KUKA KRL program: style1drop1opt2AutoRR.src, style1drop1opt2AutoRR.dat

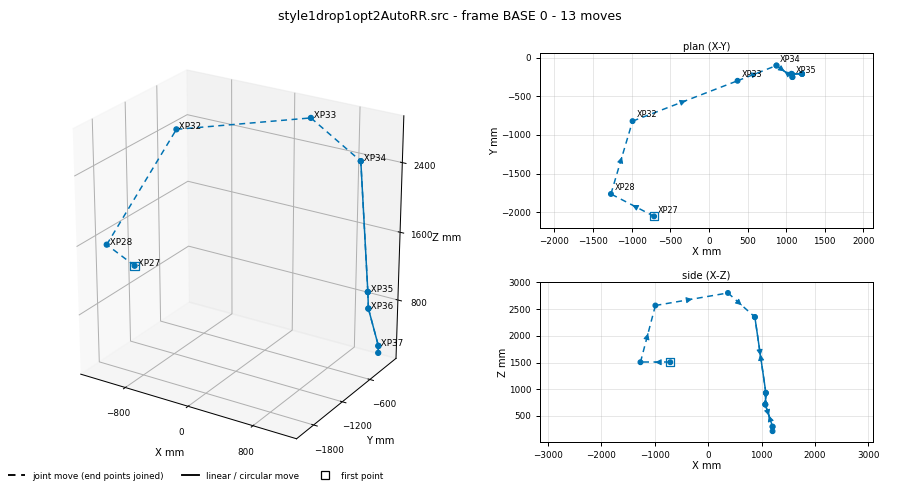
[picture p0: tool path of style1drop1opt2AutoRR.src in frame BASE 0, 13 of 14 moves have a stored position in this frame; points joined in program order, loops and branches not executed]
--- style1drop1opt2AutoRR.src ---
&ACCESS RVO1
&REL 269
&COMMENT 03-10-R1 RED RABBIT DROP
&PARAM EDITMASK = *
&PARAM DISKPATH = KRC:\R1\Program\StyleDrops\Options
DEF style1drop1opt2AutoRR( )
   ;FOLD INI
      ;FOLD BASISTECH INI
         GLOBAL INTERRUPT DECL 3 WHEN $STOPMESS==TRUE DO IR_STOPM ( )
         INTERRUPT ON 3
         BAS (#INITMOV,0 )
      ;ENDFOLD (BASISTECH INI)
      ;FOLD USER INI
         ;Make your modifications here

      ;ENDFOLD (USER INI)
   ;ENDFOLD (INI)
;********************************
; Gestamp Standards
; Line - BMW G65 (cell 03)
; Robot 03-10-R1 (BMW-03-10-R1-MH1)
; Application - RED RABBIT DROP AT DROPOFF 2
;********************************
; CALLED BY Style1Opt10AutoRR (OPTION 12). TAKES THE RED RABBIT PART TO AtPick3 OF THIS MODULE
; AND RELEASES IT, THEN CLEARS THE RED RABBIT OUTPUTS AND THE NUT FLAGS AND RETURNS HOME.
;WARNING: GRIPPER 1 IS DRIVEN TO CLOSE AT THE START ($OUT[250] ON) AND THE RELEASE COMMAND
;  OPENS GRIPPER 3, WHICH IS INACTIVE IN grp_data.dat: GRIPPER 1 DOES NOT OPEN, THE CHECK OF
;  GRIPPER 1 OPEN THAT FOLLOWS FAILS (F19, F31)
;NOTE: THE ROBOT MOVES AWAY (LIN P23) BEFORE THE GRIPPER-EMPTY WAIT (F40)
;DROPOFF 2 REQUEST - AC_DropOffCheck(2): WAIT SIGNAL $IN[76] di076DropOffMachine2 ON
;(WAITING MESSAGE, NO TIMEOUT), THEN SIGNALS $OUT[76] do076DropOffClear2 OFF,
;$OUT[25] do025DropClearTooling OFF
;FOLD DropOff[2] Request
;FOLD ;%{h}
;Params IlfProvider=ac_zoneilf; AC_CmdZones=DropOff; AC_CmdParam=2; AC_ZoneRepo=False; AC_Blending=False
;ENDFOLD
AC_DropOffCheck (2)
;ENDFOLD

;GRIPPER 1 CLOSE (HAND-WRITTEN OUTPUTS, NO CHECK) - SIGNALS $OUT[249] do249Group1Home OFF,
;$OUT[250] do250Group1Work ON (CONTINUE: SET IN THE ADVANCE RUN)
;FOLD OUT 249 'do249Group1Home' State=FALSE CONT;%{PE}%R 8.3.43,%MKUKATPBASIS,%COUT,%VOUTX,%P 2:249, 3:do249Group1Home, 5:FALSE, 6:CONTINUE
CONTINUE
$OUT[249]=FALSE
;ENDFOLD
;FOLD OUT 250 'do250Group1Work' State=TRUE CONT;%{PE}%R 8.3.43,%MKUKATPBASIS,%COUT,%VOUTX,%P 2:250, 3:do250Group1Work, 5:TRUE, 6:CONTINUE
CONTINUE
$OUT[250]=TRUE
;ENDFOLD

;APPROACH THE RED RABBIT DROP - P27, P28, P32, P33, P34, P35, P36, P37, AtPick3
;FOLD PTP P27 Vel=100 % PDAT25 Tool[1]:TOOL 1 Base[0];%{PE}%R 8.3.43,%MKUKATPBASIS,%CMOVE,%VPTP,%P 1:PTP, 2:P27, 3:, 5:100, 7:PDAT25
$BWDSTART=FALSE
PDAT_ACT=PPDAT25
FDAT_ACT=FP27
BAS(#PTP_PARAMS,100)
PTP XP27
;ENDFOLD
;FOLD PTP P28 Vel=100 % PDAT26 Tool[1]:TOOL 1 Base[0];%{PE}%R 8.3.43,%MKUKATPBASIS,%CMOVE,%VPTP,%P 1:PTP, 2:P28, 3:, 5:100, 7:PDAT26
$BWDSTART=FALSE
PDAT_ACT=PPDAT26
FDAT_ACT=FP28
BAS(#PTP_PARAMS,100)
PTP XP28
;ENDFOLD


;FOLD PTP P32 CONT Vel=100 % PDAT30 Tool[1]:TOOL 1 Base[0];%{PE}%R 8.3.43,%MKUKATPBASIS,%CMOVE,%VPTP,%P 1:PTP, 2:P32, 3:C_DIS, 5:100, 7:PDAT30
$BWDSTART=FALSE
PDAT_ACT=PPDAT30
FDAT_ACT=FP32
BAS(#PTP_PARAMS,100)
PTP XP32 C_DIS
;ENDFOLD
;FOLD PTP P33 Vel=100 % PDAT31 Tool[1]:TOOL 1 Base[0];%{PE}%R 8.3.43,%MKUKATPBASIS,%CMOVE,%VPTP,%P 1:PTP, 2:P33, 3:, 5:100, 7:PDAT31
$BWDSTART=FALSE
PDAT_ACT=PPDAT31
FDAT_ACT=FP33
BAS(#PTP_PARAMS,100)
PTP XP33
;ENDFOLD


;FOLD PTP P34 Vel=100 % PDAT32 Tool[1]:TOOL 1 Base[0];%{PE}%R 8.3.43,%MKUKATPBASIS,%CMOVE,%VPTP,%P 1:PTP, 2:P34, 3:, 5:100, 7:PDAT32
$BWDSTART=FALSE
PDAT_ACT=PPDAT32
FDAT_ACT=FP34
BAS(#PTP_PARAMS,100)
PTP XP34
;ENDFOLD
;FOLD LIN P35 CONT Vel=2 m/s CPDAT5 Tool[1]:TOOL 1 Base[0];%{PE}%R 8.3.43,%MKUKATPBASIS,%CMOVE,%VLIN,%P 1:LIN, 2:P35, 3:C_DIS C_DIS, 5:2, 7:CPDAT5
$BWDSTART=FALSE
LDAT_ACT=LCPDAT5
FDAT_ACT=FP35
BAS(#CP_PARAMS,2)
LIN XP35 C_DIS C_DIS
;ENDFOLD
;FOLD PTP P36 CONT Vel=100 % PDAT33 Tool[1]:TOOL 1 Base[0];%{PE}%R 8.3.43,%MKUKATPBASIS,%CMOVE,%VPTP,%P 1:PTP, 2:P36, 3:C_DIS, 5:100, 7:PDAT33
$BWDSTART=FALSE
PDAT_ACT=PPDAT33
FDAT_ACT=FP36
BAS(#PTP_PARAMS,100)
PTP XP36 C_DIS
;ENDFOLD
;FOLD PTP P37 CONT Vel=100 % PDAT34 Tool[1]:TOOL 1 Base[0];%{PE}%R 8.3.43,%MKUKATPBASIS,%CMOVE,%VPTP,%P 1:PTP, 2:P37, 3:C_DIS, 5:100, 7:PDAT34
$BWDSTART=FALSE
PDAT_ACT=PPDAT34
FDAT_ACT=FP37
BAS(#PTP_PARAMS,100)
PTP XP37 C_DIS
;ENDFOLD
;FOLD LIN AtPick3 Vel=2 m/s CPDAT6 Tool[1]:TOOL 1 Base[0];%{PE}%R 8.3.43,%MKUKATPBASIS,%CMOVE,%VLIN,%P 1:LIN, 2:AtPick3, 3:, 5:2, 7:CPDAT6
$BWDSTART=FALSE
LDAT_ACT=LCPDAT6
FDAT_ACT=FAtPick3
BAS(#CP_PARAMS,2)
LIN XAtPick3
;ENDFOLD
;GRIPPER 3 OPEN - GRPg_SetStateAndCheck(3, 1, ...)
;WARNING: GRIPPER 3 IS INACTIVE IN grp_data.dat: GRIPPERTECH ONLY LOGS "GRIPPER NOT ACTIVE";
;  NO OUTPUT CHANGES AND THE PART STAYS IN THE CLOSED GRIPPER 1 (F19, F31)
;FOLD Gripper SET [3]Gripper3 State=[1]OPEN Wait 0.2[s] Check with Strategy 1 ;%{PE}
;FOLD Parameters Parameters ;%{h}
;Params IlfProvider=GripperTech.GripperSet;setgripper=3;setstate=1;setcont=nocont;waittime=0.2;errorstrategy=1
;ENDFOLD
GRPg_SetStateAndCheck(3, 1, 0.2, 1)
;ENDFOLD
;CHECK GRIPPER 1 OPEN - SIGNALS $IN[257] di257Cylinder1Home ON, $IN[258] di258Cylinder1Work OFF
;(STRATEGY 1: DIALOG IN T1/T2, STOP IN AUT/EXT - SEE THE WARNING ABOVE)
;FOLD Gripper CHECK [1]Gripper 1 State=[1]OPEN with Strategy 1 ;%{PE}
;FOLD Parameters Parameters ;%{h}
;Params IlfProvider=GripperTech.GripperCheck;setgripper=1;setstate=1;setcont=nocont;checkstrategy=1
;ENDFOLD
GRPg_Check(1, 1, FALSE, 1)
;ENDFOLD
;LEAVE THE DROP - P23 (BEFORE THE GRIPPER-EMPTY WAIT, F40)
;FOLD LIN P23 Vel=2 m/s CPDAT2 Tool[1]:TOOL 1 Base[0];%{PE}%R 8.3.43,%MKUKATPBASIS,%CMOVE,%VLIN,%P 1:LIN, 2:P23, 3:, 5:2, 7:CPDAT2
$BWDSTART=FALSE
LDAT_ACT=LCPDAT2
FDAT_ACT=FP23
BAS(#CP_PARAMS,2)
LIN XP23
;ENDFOLD
;WAIT GRIPPER EMPTY - SIGNALS $IN[253] di253PartPresent1 OFF, $IN[254] di254PartPresent2 OFF (NO TIMEOUT)
;FOLD WAIT FOR ( NOT IN 253 'di253PartPresent1' ) AND ( NOT IN 254 'di254PartPresent2' );%{PE}%R 8.3.43,%MKUKATPBASIS,%CEXT_WAIT_FOR,%VEXT_WAIT_FOR,%P 2:, 4:NOT, 5:$IN, 6:253, 7:di253PartPresent1, 9:AND, 10:, 12:NOT, 13:$IN, 14:254, 15:di254PartPresent2, 17:
WAIT FOR  (  NOT $IN[253] ) AND (  NOT $IN[254] )
;ENDFOLD

;LIN P24
;FOLD LIN P24 Vel=2 m/s CPDAT4 Tool[1]:TOOL 1 Base[0];%{PE}%R 8.3.43,%MKUKATPBASIS,%CMOVE,%VLIN,%P 1:LIN, 2:P24, 3:, 5:2, 7:CPDAT4
$BWDSTART=FALSE
LDAT_ACT=LCPDAT4
FDAT_ACT=FP24
BAS(#CP_PARAMS,2)
LIN XP24
;ENDFOLD
;PART NOT IN GRIPPER - SIGNAL $OUT[18] do018Part1InGripper OFF
;FOLD OUT 18 'do018PartInGripper1' State=FALSE ;%{PE}%R 8.3.43,%MKUKATPBASIS,%COUT,%VOUTX,%P 2:18, 3:do018PartInGripper1, 5:FALSE, 6:
$OUT[18]=FALSE
;ENDFOLD
;LEAVE - P21, P25
;FOLD LIN P21 CONT Vel=2 m/s CPDAT7 Tool[1]:TOOL 1 Base[0];%{PE}%R 8.3.43,%MKUKATPBASIS,%CMOVE,%VLIN,%P 1:LIN, 2:P21, 3:C_DIS C_DIS, 5:2, 7:CPDAT7
$BWDSTART=FALSE
LDAT_ACT=LCPDAT7
FDAT_ACT=FP21
BAS(#CP_PARAMS,2)
LIN XP21 C_DIS C_DIS
;ENDFOLD
;FOLD PTP P25 Vel=100 % PDAT23 Tool[1]:TOOL 1 Base[0];%{PE}%R 8.3.43,%MKUKATPBASIS,%CMOVE,%VPTP,%P 1:PTP, 2:P25, 3:, 5:100, 7:PDAT23
$BWDSTART=FALSE
PDAT_ACT=PPDAT23
FDAT_ACT=FP25
BAS(#PTP_PARAMS,100)
PTP XP25
;ENDFOLD

;DROPOFF 2 CLEAR - AC_DropOff(2,TRUE): SIGNAL $OUT[76] do076DropOffClear2 ON; THEN RED RABBIT
;OUTPUTS OFF - SIGNALS $OUT[141] do141RedRabbitFailed OFF, $OUT[142] do142RedRabbitPassed OFF -
;AND PARTPRESENT1..3 = FALSE
;WARNING: THE RESETS WERE TYPED BY HAND INSIDE THE INLINE FORM - CONFIRMING THE FORM DELETES
;  THEM (F32). THE RESULT IS CLEARED BEFORE THE PLC CAN READ IT AT THE END OF THE CYCLE (F19)
;FOLD DropOff[2] Reset
;FOLD ;%{h}
;Params IlfProvider=ac_zoneilf; AC_CmdZones=DropOff; AC_CmdParam=2; AC_ZoneRepo=True; AC_Blending=False
;ENDFOLD
AC_DropOff (2,True)
do141RedRabbitFailed=FALSE
do142RedRabbitPassed=FALSE
PARTPRESENT1=FALSE
PARTPRESENT2=FALSE
PARTPRESENT3=FALSE
;ENDFOLD


;PTP HOME (XHOME)
;FOLD PTP HOME Vel=100 % PDAT11;%{PE}%R 8.3.43,%MKUKATPBASIS,%CMOVE,%VPTP,%P 1:PTP, 2:HOME, 3:, 5:100, 7:PDAT11
$BWDSTART=FALSE
PDAT_ACT=PPDAT11
FDAT_ACT=FHOME
BAS(#PTP_PARAMS,100)
$H_POS=XHOME
PTP XHOME
;ENDFOLD

END

--- style1drop1opt2AutoRR.dat ---
&ACCESS RVO1
&REL 269
&COMMENT GE4_Conveyor
&PARAM EDITMASK = *
&PARAM DISKPATH = KRC:\R1\Program\StyleDrops\Options
DEFDAT  style1drop1opt2AutoRR
;FOLD EXTERNAL DECLARATIONS;%{PE}%MKUKATPBASIS,%CEXT,%VCOMMON,%P
EXT  BAS (BAS_COMMAND  :IN,REAL  :IN )
DECL INT SUCCESS
;ENDFOLD (BASISTECH EXT)
;FOLD USER EXT;%{E}%MKUKATPUSER,%CEXT,%VEXT,%P
;Make here your modifications

;ENDFOLD (USER EXT)
;ENDFOLD (EXTERNAL DECLARATIONS)
DECL BASIS_SUGG_T LAST_BASIS={POINT1[] "P37                     ",POINT2[] "P37                     ",CP_PARAMS[] "CPDAT6                  ",PTP_PARAMS[] "PDAT34                  ",CONT[] "                        ",CP_VEL[] "2                       ",PTP_VEL[] "100                     ",SYNC_PARAMS[] "SYNCDAT                 ",SPL_NAME[] "S0                      ",A_PARAMS[] "ADAT0                   "}
DECL MODULEPARAM_T LAST_TP_PARAMS={PARAMS[] "AC_CmdZones=DropOff; AC_CmdParam=2; AC_ZoneRepo=True; AC_UseState=True; AC_Blending=False                               "}
DECL PDAT PPDAT11={VEL 100.000,ACC 100.000,APO_DIST 100.000,GEAR_JERK 50.0000,EXAX_IGN 0}
DECL E6POS XP21={X 1081.09485,Y -250.197342,Z 931.476,A -96.8303,B 37.9899406,C -15.7576666,S 2,T 3,E1 0.0,E2 0.0,E3 0.0,E4 0.0,E5 0.0,E6 0.0}
DECL FDAT FP21={TOOL_NO 1,BASE_NO 0,IPO_FRAME #BASE,POINT2[] " ",TQ_STATE FALSE}
DECL E6POS XP23={X 1206.28552,Y -208.912079,Z 298.869293,A -91.4409,B -0.232810885,C 0.168288454,S 2,T 3,E1 0.0,E2 0.0,E3 0.0,E4 0.0,E5 0.0,E6 0.0}
DECL FDAT FP23={TOOL_NO 1,BASE_NO 0,IPO_FRAME #BASE,POINT2[] " ",TQ_STATE FALSE}
DECL LDAT LCPDAT2={VEL 2.00000,ACC 100.000,APO_DIST 100.000,APO_FAC 50.0000,AXIS_VEL 100.000,AXIS_ACC 100.000,ORI_TYP #VAR,CIRC_TYP #BASE,JERK_FAC 50.0000,GEAR_JERK 50.0000,EXAX_IGN 0}
DECL E6POS XP24={X 1070.58411,Y -208.124802,Z 713.745911,A -91.4409,B -0.232811436,C 0.168283015,S 2,T 3,E1 0.0,E2 0.0,E3 0.0,E4 0.0,E5 0.0,E6 0.0}
DECL FDAT FP24={TOOL_NO 1,BASE_NO 0,IPO_FRAME #BASE,POINT2[] " ",TQ_STATE FALSE}
DECL LDAT LCPDAT4={VEL 2.00000,ACC 100.000,APO_DIST 100.000,APO_FAC 50.0000,AXIS_VEL 100.000,AXIS_ACC 100.000,ORI_TYP #VAR,CIRC_TYP #BASE,JERK_FAC 50.0000,GEAR_JERK 50.0000,EXAX_IGN 0}
DECL E6POS XP25={X 874.811584,Y -100.693466,Z 2352.82349,A -4.40710449,B 2.42972946,C 0.669244647,S 2,T 10,E1 0.0,E2 0.0,E3 0.0,E4 0.0,E5 0.0,E6 0.0}
DECL FDAT FP25={TOOL_NO 1,BASE_NO 0,IPO_FRAME #BASE,POINT2[] " ",TQ_STATE FALSE}
DECL PDAT PPDAT23={VEL 100.000,ACC 100.000,APO_DIST 100.000,APO_MODE #CDIS,GEAR_JERK 50.0000,EXAX_IGN 0}
DECL E6POS XP27={X -709.692566,Y -2053.68652,Z 1506.28467,A -104.821503,B 4.90587568,C 179.018478,S 2,T 34,E1 0.0,E2 0.0,E3 0.0,E4 0.0,E5 0.0,E6 0.0}
DECL FDAT FP27={TOOL_NO 1,BASE_NO 0,IPO_FRAME #BASE,POINT2[] " ",TQ_STATE FALSE}
DECL PDAT PPDAT25={VEL 100.000,ACC 100.000,APO_DIST 100.000,APO_MODE #CDIS,GEAR_JERK 50.0000,EXAX_IGN 0}
DECL E6POS XP28={X -1268.63135,Y -1764.04834,Z 1506.28467,A -121.480026,B 4.90587568,C 179.018478,S 2,T 34,E1 0.0,E2 0.0,E3 0.0,E4 0.0,E5 0.0,E6 0.0}
DECL FDAT FP28={TOOL_NO 1,BASE_NO 0,IPO_FRAME #BASE,POINT2[] " ",TQ_STATE FALSE}
DECL PDAT PPDAT26={VEL 100.000,ACC 100.000,APO_DIST 100.000,APO_MODE #CDIS,GEAR_JERK 50.0000,EXAX_IGN 0}
DECL PDAT PPDAT30={VEL 100.000,ACC 100.000,APO_DIST 500.000,APO_MODE #CDIS,GEAR_JERK 50.0000,EXAX_IGN 0}
DECL E6POS XP32={X -988.705139,Y -820.766479,Z 2569.14844,A 137.545090,B -48.9822197,C 56.5858917,S 2,T 2,E1 0.0,E2 0.0,E3 0.0,E4 0.0,E5 0.0,E6 0.0}
DECL FDAT FP32={TOOL_NO 1,BASE_NO 0,IPO_FRAME #BASE,POINT2[] " ",TQ_STATE FALSE}
DECL PDAT PPDAT31={VEL 100.000,ACC 100.000,APO_DIST 100.000,APO_MODE #CDIS,GEAR_JERK 50.0000,EXAX_IGN 0}
DECL E6POS XP33={X 370.852905,Y -298.257416,Z 2804.38916,A -147.361786,B -35.6047363,C 79.4075775,S 2,T 2,E1 0.0,E2 0.0,E3 0.0,E4 0.0,E5 0.0,E6 0.0}
DECL FDAT FP33={TOOL_NO 1,BASE_NO 0,IPO_FRAME #BASE,POINT2[] " ",TQ_STATE FALSE}
DECL PDAT PPDAT32={VEL 100.000,ACC 100.000,APO_DIST 100.000,APO_MODE #CDIS,GEAR_JERK 50.0000,EXAX_IGN 0}
DECL E6POS XP34={X 874.811584,Y -100.693466,Z 2352.82349,A -4.40710449,B 2.42972946,C 0.669244647,S 2,T 10,E1 0.0,E2 0.0,E3 0.0,E4 0.0,E5 0.0,E6 0.0}
DECL FDAT FP34={TOOL_NO 1,BASE_NO 0,IPO_FRAME #BASE,POINT2[] " ",TQ_STATE FALSE}
DECL LDAT LCPDAT5={VEL 2.00000,ACC 100.000,APO_DIST 100.000,APO_FAC 50.0000,AXIS_VEL 100.000,AXIS_ACC 100.000,ORI_TYP #VAR,CIRC_TYP #BASE,JERK_FAC 50.0000,GEAR_JERK 50.0000,EXAX_IGN 0}
DECL E6POS XP35={X 1081.09485,Y -250.197342,Z 931.476,A -96.8303,B 37.9899406,C -15.7576666,S 2,T 3,E1 0.0,E2 0.0,E3 0.0,E4 0.0,E5 0.0,E6 0.0}
DECL FDAT FP35={TOOL_NO 1,BASE_NO 0,IPO_FRAME #BASE,POINT2[] " ",TQ_STATE FALSE}
DECL PDAT PPDAT33={VEL 100.000,ACC 100.000,APO_DIST 500.000,APO_MODE #CDIS,GEAR_JERK 50.0000,EXAX_IGN 0}
DECL E6POS XP36={X 1070.46545,Y -208.124084,Z 714.012268,A -91.4409,B -0.232809603,C 0.168291062,S 2,T 3,E1 0.0,E2 0.0,E3 0.0,E4 0.0,E5 0.0,E6 0.0}
DECL FDAT FP36={TOOL_NO 1,BASE_NO 0,IPO_FRAME #BASE,POINT2[] " ",TQ_STATE FALSE}
DECL PDAT PPDAT34={VEL 100.000,ACC 100.000,APO_DIST 10.0000,APO_MODE #CDIS,GEAR_JERK 50.0000,EXAX_IGN 0}
DECL E6POS XP37={X 1206.28552,Y -208.912048,Z 298.869263,A -91.4409,B -0.232809111,C 0.168290,S 2,T 3,E1 0.0,E2 0.0,E3 0.0,E4 0.0,E5 0.0,E6 0.0}
DECL FDAT FP37={TOOL_NO 1,BASE_NO 0,IPO_FRAME #BASE,POINT2[] " ",TQ_STATE FALSE}
DECL LDAT LCPDAT6={VEL 2.00000,ACC 100.000,APO_DIST 0.0,APO_FAC 50.0000,AXIS_VEL 100.000,AXIS_ACC 100.000,ORI_TYP #VAR,CIRC_TYP #BASE,JERK_FAC 50.0000,GEAR_JERK 50.0000,EXAX_IGN 0}
DECL E6POS XAtPick3={X 1206.28552,Y -208.912048,Z 214.158249,A -91.4409,B -0.232809141,C 0.168289974,S 2,T 3,E1 0.0,E2 0.0,E3 0.0,E4 0.0,E5 0.0,E6 0.0}
DECL FDAT FAtPick3={TOOL_NO 1,BASE_NO 0,IPO_FRAME #BASE,POINT2[] " ",TQ_STATE FALSE}
DECL LDAT LCPDAT7={VEL 2.00000,ACC 100.000,APO_DIST 100.000,APO_FAC 50.0000,AXIS_VEL 100.000,AXIS_ACC 100.000,ORI_TYP #VAR,CIRC_TYP #BASE,JERK_FAC 50.0000,GEAR_JERK 50.0000,EXAX_IGN 0}
ENDDAT
